(* CoDeSys 2.3.5.6 project: egzamin.pro *)
(* Libraries: Standard.lib 4.1.15 17:23:13, SYSLIBCALLBACK.LIB 4.1.15 17:23:13 *)

(* PLC configuration (modules and I/O channels)
Local I/O [EC4P_LocalIO] node 0, in %IB0 out %QB0 {EC4P_LocalInt = 0}
  I1 AT %IX0.0 [LocalBitInput] Input I1
  I2 AT %IX0.1 [LocalBitInput] Input I2
  I3 AT %IX0.2 [LocalBitInput] Input I3
  I4 AT %IX0.3 [LocalBitInput] Input I4
  I5 AT %IX0.4 [LocalBitInput] Input I5
  I6 AT %IX0.5 [LocalBitInput] Input I6
  I7 AT %IX0.6 [LocalBitInput] Input I7
  I8 AT %IX0.7 [LocalBitInput] Input I8
  I9 AT %IX1.0 [LocalBitInput] Input I9
  I10 AT %IX1.1 [LocalBitInput] Input I10
  I11 AT %IX1.2 [LocalBitInput] Input I11
  I12 AT %IX1.3 [LocalBitInput] Input I12
  I13 AT %IX1.4 [LocalDiagInput] Diagnostic Input I13
  I14 AT %IX1.5 [LocalDiagInput] Diagnostic Input I14
  I15 AT %IX1.6 [LocalDiagInput] Diagnostic Input I15
  I16 AT %IX1.7 [LocalDiagInput] Diagnostic Input I16
  I7_Analog AT %IW2 [LocalAnalogIn] Input I7, 10Bit, 0-10VDC
  I8_Analog AT %IW4 [LocalAnalogIn] Input I8, 10Bit, 0-10VDC
  I11_Analog AT %IW6 [LocalAnalogIn] Input I11, 10Bit, 0-10VDC
  I12_Analog AT %IW8 [LocalAnalogIn] Input I12, 10Bit, 0-10VDC
  Transistor Outputs [EC4P_TOutputs] node 0, in %IB10 out %QB0
    Q1 AT %QX0.0 [LocalBitOutput] Transistor-Output Q1
    Q2 AT %QX0.1 [LocalBitOutput] Transistor-Output Q2
    Q3 AT %QX0.2 [LocalBitOutput] Transistor-Output Q3
    Q4 AT %QX0.3 [LocalBitOutput] Transistor-Output Q4
    Q5 AT %QX0.4 [LocalBitOutput] Transistor-Output Q5
    Q6 AT %QX0.5 [LocalBitOutput] Transistor-Output Q6
    Q7 AT %QX0.6 [LocalBitOutput] Transistor-Output Q7
    Q8 AT %QX0.7 [LocalBitOutput] Transistor-Output Q8
  No Analog Output [EC4P_NoAnalogOutput] node 1, in %IB10 out %QB1
  No Keys [EC4P_NoKeys] node 2, in %IB10 out %QB1
  No Counter [EC4P_NoCounter] node 3, in %IB10 out %QB1
Extension [EC4P_Extension] node 1, in %IB10 out %QB1
  No Extension [EC4P_NoExtension] node 0, in %IB10 out %QB1
*)

(* POU PLC_PRG, CFC *)
PROGRAM PLC_PRG
VAR
	TP1: TP;
	TP2: TP;
	ON: BOOL;
	TTP1: TIME;
	FTRIG1: F_TRIG;
	TTP2: TIME;
END_VAR
VAR (* helpers for the ST form of the networks *)
	_t428 : BOOL;
END_VAR
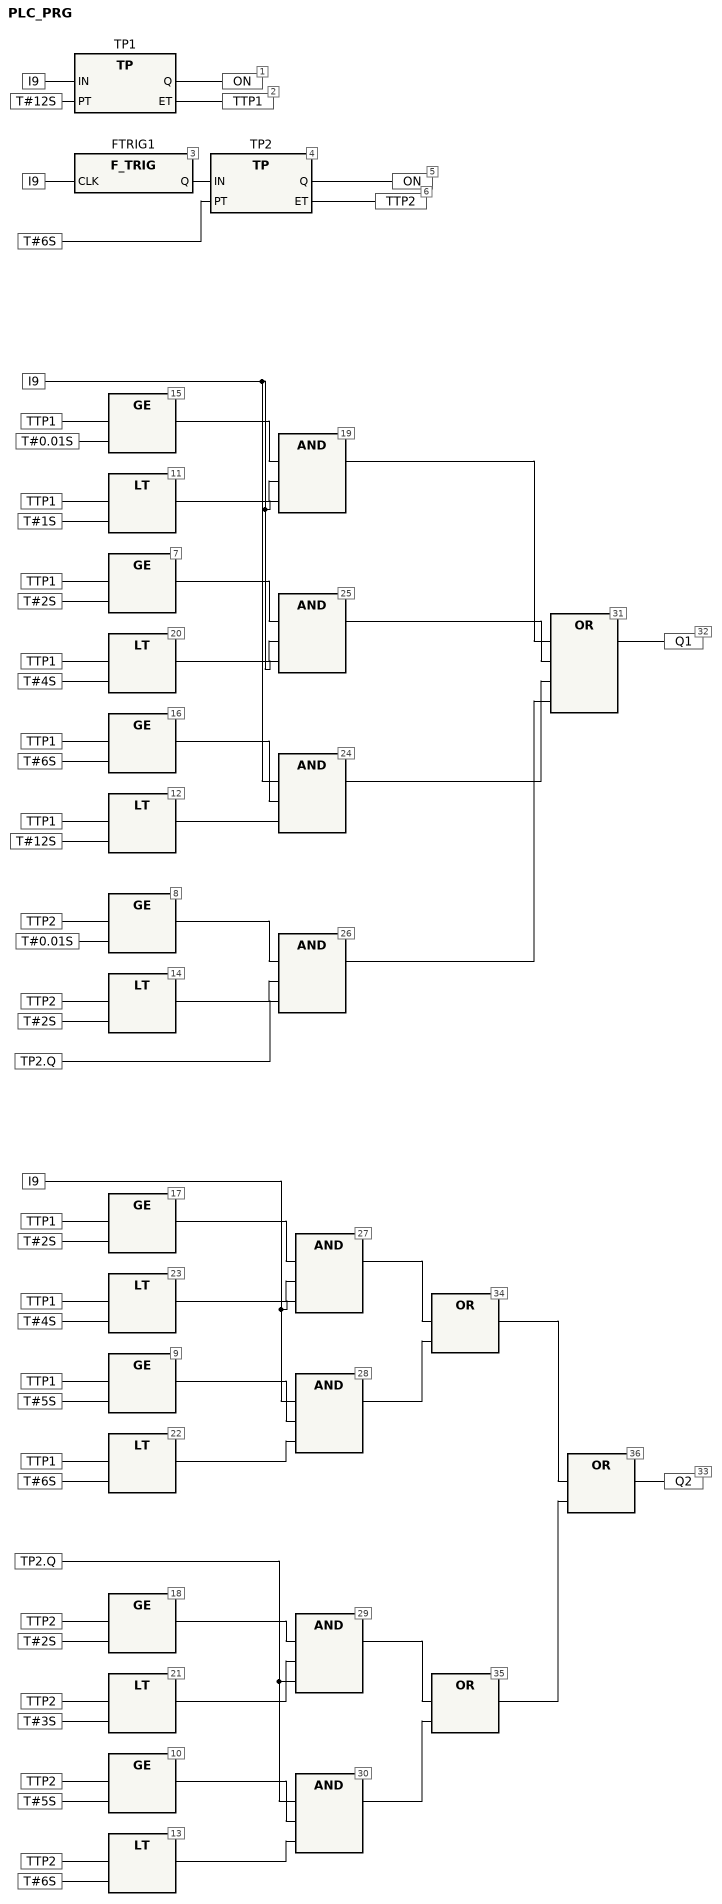
_CFC_ (* Continuous Function Chart, elements in execution order *)
#0 TP1:TP(IN: I9, PT: T#12S)
#1 ON <= #0.Q
#2 TTP1 <= #0.ET
#3 FTRIG1:F_TRIG(CLK: I9)
#4 TP2:TP(IN: #3.Q, PT: T#6S)
#5 ON <= #4.Q
#6 TTP2 <= #4.ET
#7 GE(TTP1, T#2S)
#8 GE(TTP2, T#0.01S)
#9 GE(TTP1, T#5S)
#10 GE(TTP2, T#5S)
#11 LT(TTP1, T#1S)
#12 LT(TTP1, T#12S)
#13 LT(TTP2, T#6S)
#14 LT(TTP2, T#2S)
#15 GE(TTP1, T#0.01S)
#16 GE(TTP1, T#6S)
#17 GE(TTP1, T#2S)
#18 GE(TTP2, T#2S)
#19 AND(#15, #11, I9)
#20 LT(TTP1, T#4S)
#21 LT(TTP2, T#3S)
#22 LT(TTP1, T#6S)
#23 LT(TTP1, T#4S)
#24 AND(I9, #16, #12)
#25 AND(#7, #20, I9)
#26 AND(#8, #14, TP2.Q)
#27 AND(#17, #23, I9)
#28 AND(I9, #9, #22)
#29 AND(#18, #21, TP2.Q)
#30 AND(TP2.Q, #10, #13)
#31 OR(#19, #25, #24, #26)
#32 Q1 <= #31
#33 Q2 <= #36
#34 OR(#27, #28)
#35 OR(#29, #30)
#36 OR(#34, #35)
_END_CFC_
(* the same logic as Structured Text *)
TP1(IN := I9, PT := T#12S);
ON := TP1.Q;
TTP1 := TP1.ET;
FTRIG1(CLK := I9);
TP2(IN := FTRIG1.Q, PT := T#6S);
ON := TP2.Q;
TTP2 := TP2.ET;
Q1 := ((TTP1 >= T#0.01S) AND (TTP1 < T#1S) AND I9) OR ((TTP1 >= T#2S) AND (TTP1 < T#4S) AND I9) OR (I9 AND (TTP1 >= T#6S) AND (TTP1 < T#12S)) OR ((TTP2 >= T#0.01S) AND (TTP2 < T#2S) AND TP2.Q);
Q2 := _t428;
_t428 := (((TTP1 >= T#2S) AND (TTP1 < T#4S) AND I9) OR (I9 AND (TTP1 >= T#5S) AND (TTP1 < T#6S))) OR (((TTP2 >= T#2S) AND (TTP2 < T#3S) AND TP2.Q) OR (TP2.Q AND (TTP2 >= T#5S) AND (TTP2 < T#6S)));
END_PROGRAM
